SUBAPPLICATION Uebung_HystereseHorizontal_AX_simple (* MID/DEAD/HYSTERESIS-Eingabefelder bewegen live die 5 Schwellwert-Dreiecke im horizontalen Bargraph (wie Uebung_225_AX fuer Workspace_Dreieck, aber 5 Marker statt 1 und mit AR-Arithmetik fuer die 4 abgeleiteten Schwellen) *)
  (* Standard: 61499-2; Description: Copyright (c) 2026 Meisterschulen am Ostbahnhof This program and the accompanying materials are made available under the terms of the Eclipse Public License 2.0 which is available at https://www.eclipse.org/legal/epl-2.0/ SPDX-License-Identifier: EPL-2.0 *)
  (* Version 1.1, 2026-09-27, Franz Höpfinger, Meisterschulen am Ostbahnhof, AR_TO_AI, Zero, QPos zu MyLib::sys::Q_ChildPosition_AR_Horizontal SubApp ausgelagert *)
  PACKAGE Uebungen;
  IMPORT Uebungen::const::UT::HystereseHorizontal::DefaultPool_Numeric::InputNumber_MID_N;
  IMPORT Uebungen::const::UT::HystereseHorizontal::DefaultPool_Numeric::InputNumber_DEAD_N;
  IMPORT Uebungen::const::UT::HystereseHorizontal::DefaultPool_Numeric::InputNumber_HYSTERESIS_N;
  IMPORT Uebungen::const::UT::HystereseHorizontal::DefaultPool::Polygon_MID;
  IMPORT Uebungen::const::UT::HystereseHorizontal::DefaultPool::Polygon_MID_PLUS_DEAD;
  IMPORT Uebungen::const::UT::HystereseHorizontal::DefaultPool::Polygon_MID_MINUS_DEAD;
  IMPORT Uebungen::const::UT::HystereseHorizontal::DefaultPool::Polygon_MID_PLUS_DEAD_HYST;
  IMPORT Uebungen::const::UT::HystereseHorizontal::DefaultPool::Polygon_MID_MINUS_DEAD_HYST;
  IMPORT Uebungen::const::UT::HystereseHorizontal::DefaultPool::Container_Schwellwerte;
  IMPORT Uebungen::const::UT::HystereseHorizontal::DefaultPool_Bargraph::Bargraph_Hysterese_ScalePx;
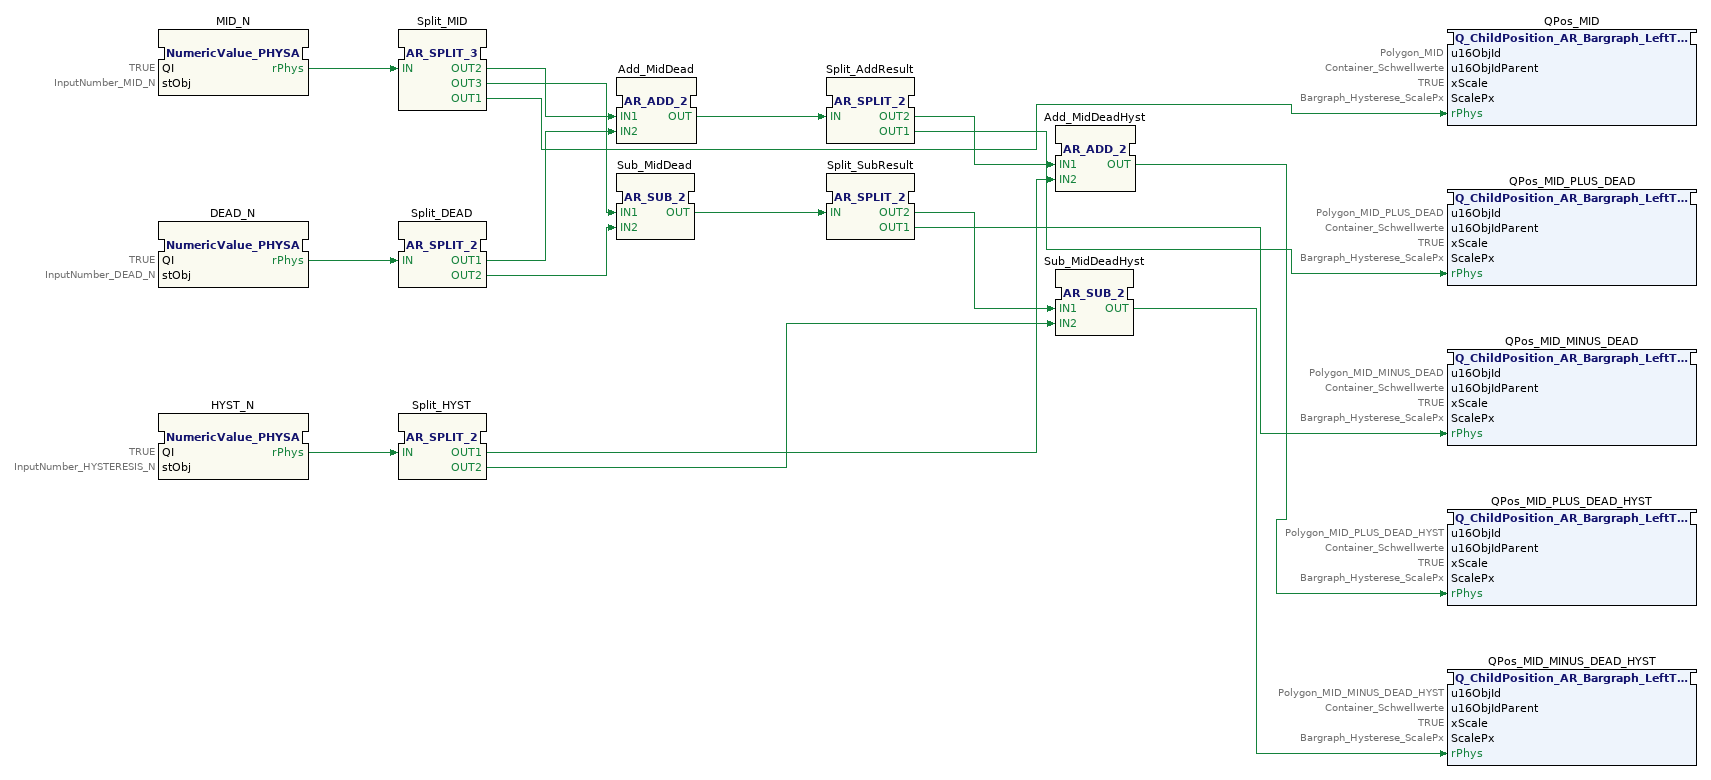
  FBS
    MID_N : isobus::UT::io::NumericValue::NumericValue_PHYSA(QI := TRUE, stObj := InputNumber_MID_N);
    DEAD_N : isobus::UT::io::NumericValue::NumericValue_PHYSA(QI := TRUE, stObj := InputNumber_DEAD_N);
    HYST_N : isobus::UT::io::NumericValue::NumericValue_PHYSA(QI := TRUE, stObj := InputNumber_HYSTERESIS_N);
    Split_MID : adapter::events::unidirectional::AR_SPLIT_3;
    Split_DEAD : adapter::events::unidirectional::AR_SPLIT_2;
    Split_HYST : adapter::events::unidirectional::AR_SPLIT_2;
    Add_MidDead : adapter::iec61131::arithmetic::AR_ADD_2;
    Sub_MidDead : adapter::iec61131::arithmetic::AR_SUB_2;
    Split_AddResult : adapter::events::unidirectional::AR_SPLIT_2;
    Split_SubResult : adapter::events::unidirectional::AR_SPLIT_2;
    Add_MidDeadHyst : adapter::iec61131::arithmetic::AR_ADD_2;
    Sub_MidDeadHyst : adapter::iec61131::arithmetic::AR_SUB_2;
  END_FBS
  SUBAPPS
    QPos_MID : MyLib::sys::Q_ChildPosition_AR_Bargraph_LeftToRight(u16ObjId := Polygon_MID, u16ObjIdParent := Container_Schwellwerte, xScale := TRUE, ScalePx := Bargraph_Hysterese_ScalePx);
    QPos_MID_PLUS_DEAD : MyLib::sys::Q_ChildPosition_AR_Bargraph_LeftToRight(u16ObjId := Polygon_MID_PLUS_DEAD, u16ObjIdParent := Container_Schwellwerte, xScale := TRUE, ScalePx := Bargraph_Hysterese_ScalePx);
    QPos_MID_MINUS_DEAD : MyLib::sys::Q_ChildPosition_AR_Bargraph_LeftToRight(u16ObjId := Polygon_MID_MINUS_DEAD, u16ObjIdParent := Container_Schwellwerte, xScale := TRUE, ScalePx := Bargraph_Hysterese_ScalePx);
    QPos_MID_PLUS_DEAD_HYST : MyLib::sys::Q_ChildPosition_AR_Bargraph_LeftToRight(u16ObjId := Polygon_MID_PLUS_DEAD_HYST, u16ObjIdParent := Container_Schwellwerte, xScale := TRUE, ScalePx := Bargraph_Hysterese_ScalePx);
    QPos_MID_MINUS_DEAD_HYST : MyLib::sys::Q_ChildPosition_AR_Bargraph_LeftToRight(u16ObjId := Polygon_MID_MINUS_DEAD_HYST, u16ObjIdParent := Container_Schwellwerte, xScale := TRUE, ScalePx := Bargraph_Hysterese_ScalePx);
  END_SUBAPPS
  ADAPTER_CONNECTIONS
    MID_N.rPhys TO Split_MID.IN;
    DEAD_N.rPhys TO Split_DEAD.IN;
    HYST_N.rPhys TO Split_HYST.IN;
    Split_MID.OUT2 TO Add_MidDead.IN1;
    Split_DEAD.OUT1 TO Add_MidDead.IN2;
    Split_MID.OUT3 TO Sub_MidDead.IN1;
    Split_DEAD.OUT2 TO Sub_MidDead.IN2;
    Add_MidDead.OUT TO Split_AddResult.IN;
    Sub_MidDead.OUT TO Split_SubResult.IN;
    Split_AddResult.OUT2 TO Add_MidDeadHyst.IN1;
    Split_HYST.OUT1 TO Add_MidDeadHyst.IN2;
    Split_SubResult.OUT2 TO Sub_MidDeadHyst.IN1;
    Split_HYST.OUT2 TO Sub_MidDeadHyst.IN2;
    Split_MID.OUT1 TO QPos_MID.rPhys;
    Split_AddResult.OUT1 TO QPos_MID_PLUS_DEAD.rPhys;
    Split_SubResult.OUT1 TO QPos_MID_MINUS_DEAD.rPhys;
    Add_MidDeadHyst.OUT TO QPos_MID_PLUS_DEAD_HYST.rPhys;
    Sub_MidDeadHyst.OUT TO QPos_MID_MINUS_DEAD_HYST.rPhys;
  END_CONNECTIONS
END_SUBAPPLICATION
